SUBAPPLICATION Uebung_014 (* Container (visible/invisible) *)
  (* Standard: 61499-2; Description: Copyright (c) 2023 Meisterschulen am Ostbahnhof This program and the accompanying materials are made available under the terms of the Eclipse Public License 2.0 which is available at https://www.eclipse.org/legal/epl-2.0/ SPDX-License-Identifier: EPL-2.0 *)
  (* Version 1.0, 2023-10-23, Franz Höpfinger, Meisterschulen am Ostbahnhof *)
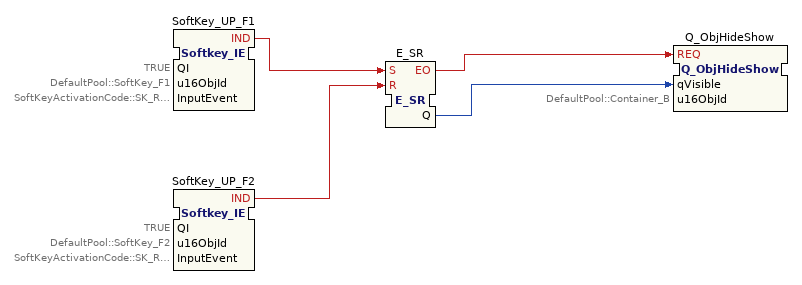
  FBS
    SoftKey_UP_F1 : Softkey_IE(QI := TRUE, u16ObjId := DefaultPool::SoftKey_F1, InputEvent := SoftKeyActivationCode::SK_RELEASED);
    SoftKey_UP_F2 : Softkey_IE(QI := TRUE, u16ObjId := DefaultPool::SoftKey_F2, InputEvent := SoftKeyActivationCode::SK_RELEASED);
    E_SR : iec61499::events::E_SR;
    Q_ObjHideShow : isobus::ut::Q_ObjHideShow(u16ObjId := DefaultPool::Container_B);
  END_FBS
  EVENT_CONNECTIONS
    SoftKey_UP_F1.IND TO E_SR.S;
    SoftKey_UP_F2.IND TO E_SR.R;
    E_SR.EO TO Q_ObjHideShow.REQ;
  END_CONNECTIONS
  DATA_CONNECTIONS
    E_SR.Q TO Q_ObjHideShow.qVisible;
  END_CONNECTIONS
END_SUBAPPLICATION
